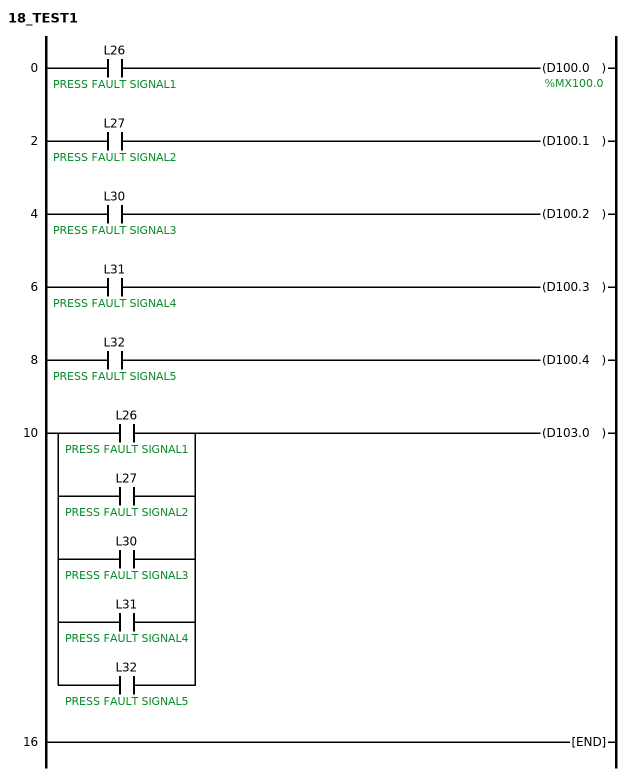
[picture p312: ladder of 18_TEST1, rungs at steps 0 to 16]
0     LD      L26  ; PRESS FAULT SIGNAL1
      OUT     D100.0  ; %MX100.0
2     LD      L27  ; PRESS FAULT SIGNAL2
      OUT     D100.1
4     LD      L30  ; PRESS FAULT SIGNAL3
      OUT     D100.2
6     LD      L31  ; PRESS FAULT SIGNAL4
      OUT     D100.3
8     LD      L32  ; PRESS FAULT SIGNAL5
      OUT     D100.4
10    LD      L26  ; PRESS FAULT SIGNAL1
      OR      L27  ; PRESS FAULT SIGNAL2
      OR      L30  ; PRESS FAULT SIGNAL3
      OR      L31  ; PRESS FAULT SIGNAL4
      OR      L32  ; PRESS FAULT SIGNAL5
      OUT     D103.0
16    END
END_PROGRAM

PROGRAM Map
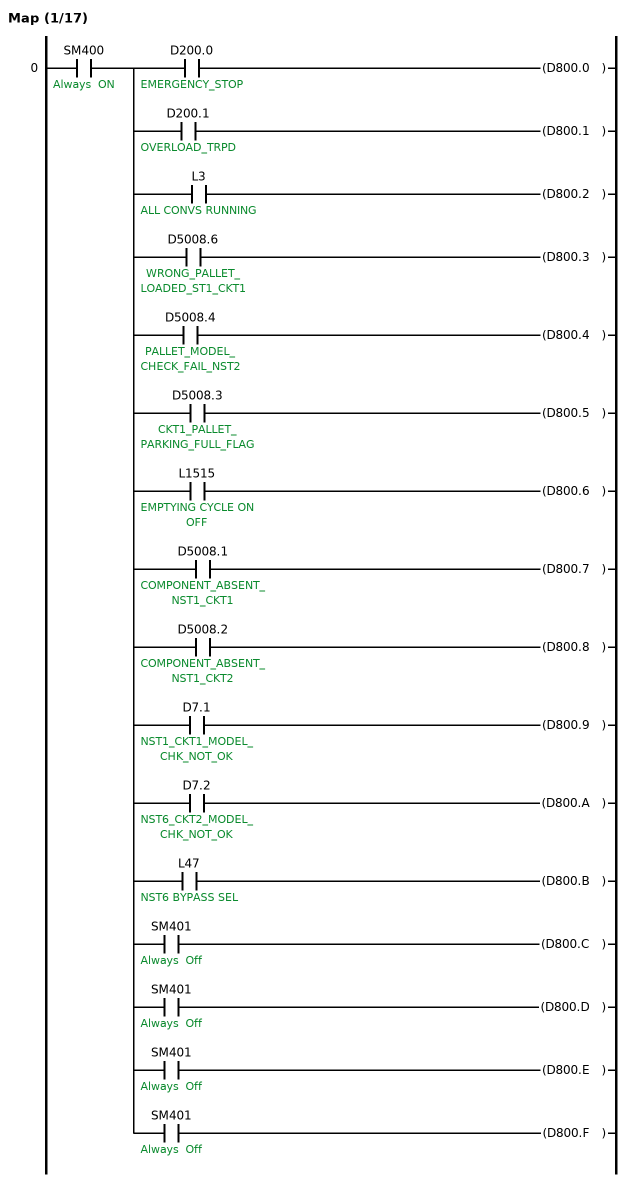
0     LD      SM400  ; Always  ON
      MPS
      AND     D200.0  ; EMERGENCY_STOP
      OUT     D800.0
      MRD
      AND     D200.1  ; OVERLOAD_TRPD
      OUT     D800.1
      MRD
      AND     L3  ; ALL CONVS RUNNING
      OUT     D800.2
      MRD
      AND     D5008.6  ; WRONG_PALLET_LOADED_ST1_CKT1
      OUT     D800.3
      MRD
      AND     D5008.4  ; PALLET_MODEL_CHECK_FAIL_NST2
      OUT     D800.4
      MRD
      AND     D5008.3  ; CKT1_PALLET_PARKING_FULL_FLAG
      OUT     D800.5
      MRD
      AND     L1515  ; EMPTYING CYCLE ON OFF
      OUT     D800.6
      MRD
      AND     D5008.1  ; COMPONENT_ABSENT_NST1_CKT1
      OUT     D800.7
      MRD
      AND     D5008.2  ; COMPONENT_ABSENT_NST1_CKT2
      OUT     D800.8
      MRD
      AND     D7.1  ; NST1_CKT1_MODEL_CHK_NOT_OK
      OUT     D800.9
      MRD
      AND     D7.2  ; NST6_CKT2_MODEL_CHK_NOT_OK
      OUT     D800.A
      MRD
      AND     L47  ; NST6 BYPASS SEL
      OUT     D800.B
      MRD
      AND     SM401  ; Always  Off
      OUT     D800.C
      MRD
      AND     SM401  ; Always  Off
      OUT     D800.D
      MRD
      AND     SM401  ; Always  Off
      OUT     D800.E
      MPP
      AND     SM401  ; Always  Off
      OUT     D800.F
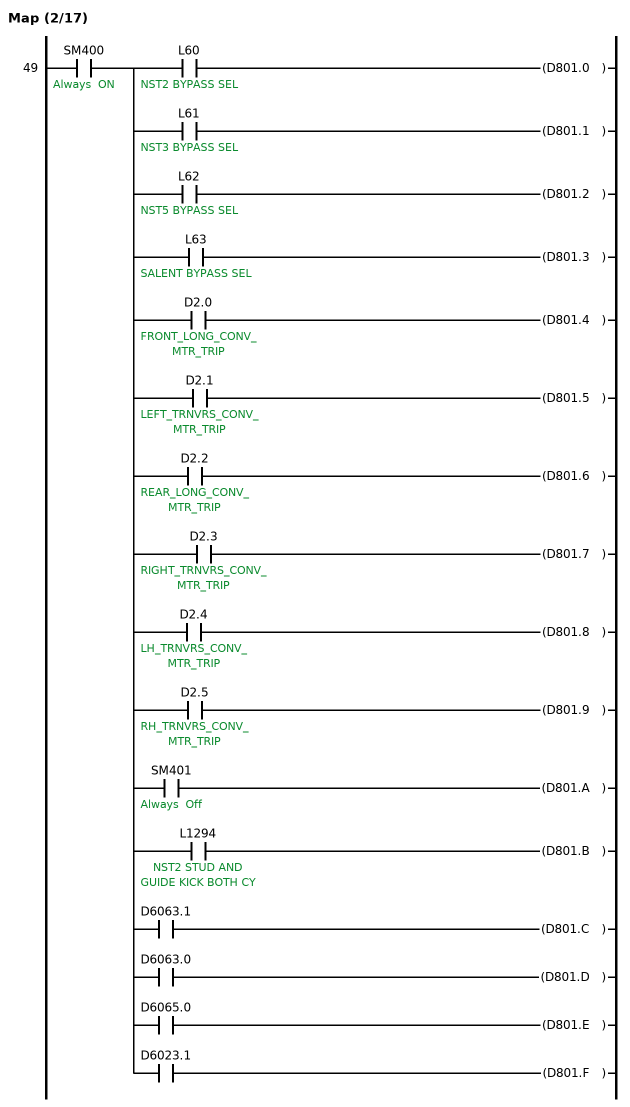
49    LD      SM400  ; Always  ON
      MPS
      AND     L60  ; NST2 BYPASS SEL
      OUT     D801.0
      MRD
      AND     L61  ; NST3 BYPASS SEL
      OUT     D801.1
      MRD
      AND     L62  ; NST5 BYPASS SEL
      OUT     D801.2
      MRD
      AND     L63  ; SALENT BYPASS SEL
      OUT     D801.3
      MRD
      AND     D2.0  ; FRONT_LONG_CONV_MTR_TRIP
      OUT     D801.4
      MRD
      AND     D2.1  ; LEFT_TRNVRS_CONV_MTR_TRIP
      OUT     D801.5
      MRD
      AND     D2.2  ; REAR_LONG_CONV_MTR_TRIP
      OUT     D801.6
      MRD
      AND     D2.3  ; RIGHT_TRNVRS_CONV_MTR_TRIP
      OUT     D801.7
      MRD
      AND     D2.4  ; LH_TRNVRS_CONV_MTR_TRIP
      OUT     D801.8
      MRD
      AND     D2.5  ; RH_TRNVRS_CONV_MTR_TRIP
      OUT     D801.9
      MRD
      AND     SM401  ; Always  Off
      OUT     D801.A
      MRD
      AND     L1294  ; NST2 STUD AND GUIDE KICK BOTH CY
      OUT     D801.B
      MRD
      AND     D6063.1
      OUT     D801.C
      MRD
      AND     D6063.0
      OUT     D801.D
      MRD
      AND     D6065.0
      OUT     D801.E
      MPP
      AND     D6023.1
      OUT     D801.F
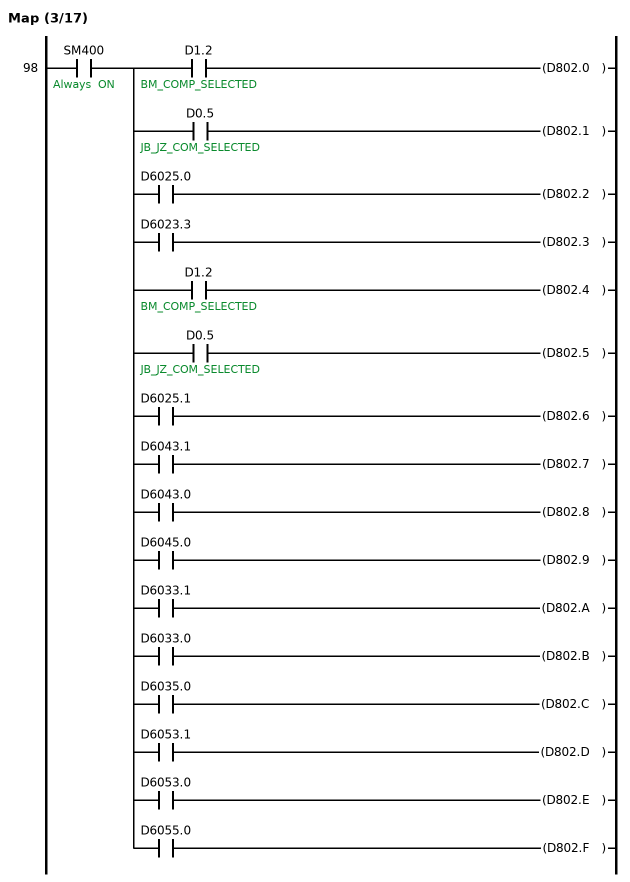
98    LD      SM400  ; Always  ON
      MPS
      AND     D1.2  ; BM_COMP_SELECTED
      OUT     D802.0
      MRD
      AND     D0.5  ; JB_JZ_COM_SELECTED
      OUT     D802.1
      MRD
      AND     D6025.0
      OUT     D802.2
      MRD
      AND     D6023.3
      OUT     D802.3
      MRD
      AND     D1.2  ; BM_COMP_SELECTED
      OUT     D802.4
      MRD
      AND     D0.5  ; JB_JZ_COM_SELECTED
      OUT     D802.5
      MRD
      AND     D6025.1
      OUT     D802.6
      MRD
      AND     D6043.1
      OUT     D802.7
      MRD
      AND     D6043.0
      OUT     D802.8
      MRD
      AND     D6045.0
      OUT     D802.9
      MRD
      AND     D6033.1
      OUT     D802.A
      MRD
      AND     D6033.0
      OUT     D802.B
      MRD
      AND     D6035.0
      OUT     D802.C
      MRD
      AND     D6053.1
      OUT     D802.D
      MRD
      AND     D6053.0
      OUT     D802.E
      MPP
      AND     D6055.0
      OUT     D802.F
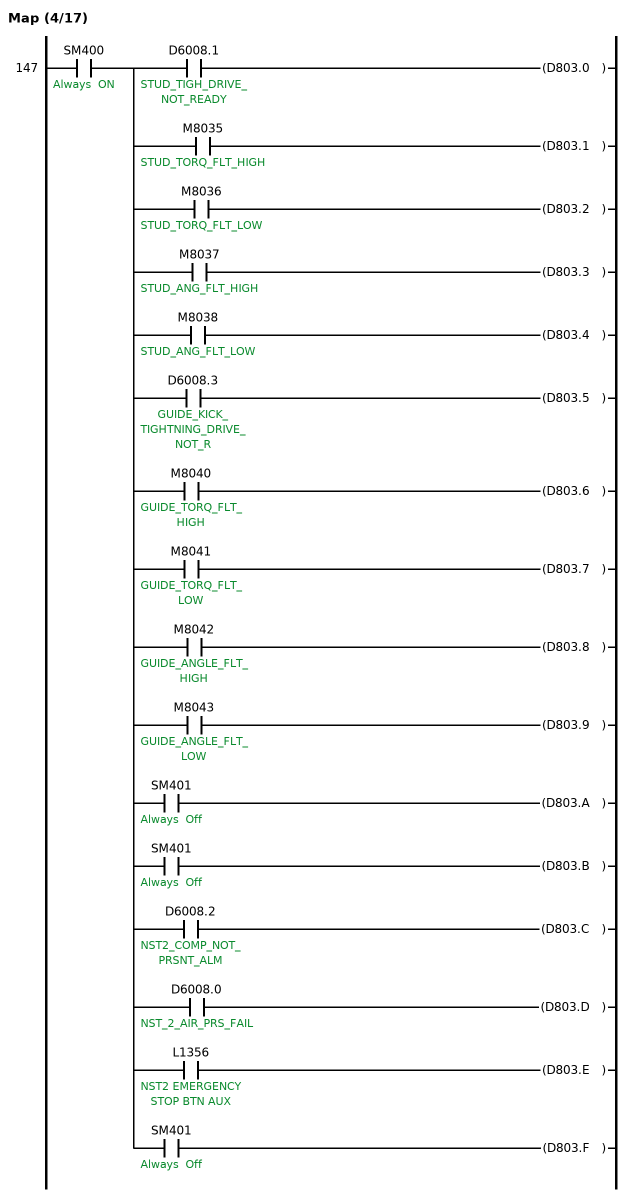
147   LD      SM400  ; Always  ON
      MPS
      AND     D6008.1  ; STUD_TIGH_DRIVE_NOT_READY
      OUT     D803.0
      MRD
      AND     M8035  ; STUD_TORQ_FLT_HIGH
      OUT     D803.1
      MRD
      AND     M8036  ; STUD_TORQ_FLT_LOW
      OUT     D803.2
      MRD
      AND     M8037  ; STUD_ANG_FLT_HIGH
      OUT     D803.3
      MRD
      AND     M8038  ; STUD_ANG_FLT_LOW
      OUT     D803.4
      MRD
      AND     D6008.3  ; GUIDE_KICK_TIGHTNING_DRIVE_NOT_R
      OUT     D803.5
      MRD
      AND     M8040  ; GUIDE_TORQ_FLT_HIGH
      OUT     D803.6
      MRD
      AND     M8041  ; GUIDE_TORQ_FLT_LOW
      OUT     D803.7
      MRD
      AND     M8042  ; GUIDE_ANGLE_FLT_HIGH
      OUT     D803.8
      MRD
      AND     M8043  ; GUIDE_ANGLE_FLT_LOW
      OUT     D803.9
      MRD
      AND     SM401  ; Always  Off
      OUT     D803.A
      MRD
      AND     SM401  ; Always  Off
      OUT     D803.B
      MRD
      AND     D6008.2  ; NST2_COMP_NOT_PRSNT_ALM
      OUT     D803.C
      MRD
      AND     D6008.0  ; NST_2_AIR_PRS_FAIL
      OUT     D803.D
      MRD
      AND     L1356  ; NST2 EMERGENCY STOP BTN AUX
      OUT     D803.E
      MPP
      AND     SM401  ; Always  Off
      OUT     D803.F
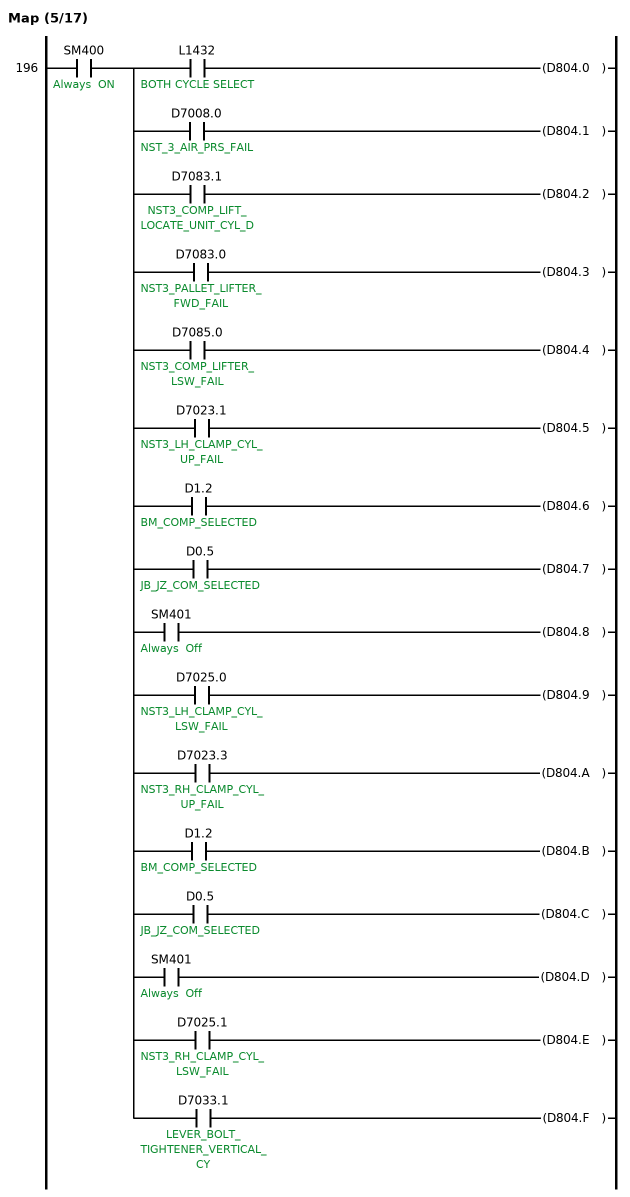
196   LD      SM400  ; Always  ON
      MPS
      AND     L1432  ; BOTH CYCLE SELECT
      OUT     D804.0
      MRD
      AND     D7008.0  ; NST_3_AIR_PRS_FAIL
      OUT     D804.1
      MRD
      AND     D7083.1  ; NST3_COMP_LIFT_LOCATE_UNIT_CYL_D
      OUT     D804.2
      MRD
      AND     D7083.0  ; NST3_PALLET_LIFTER_FWD_FAIL
      OUT     D804.3
      MRD
      AND     D7085.0  ; NST3_COMP_LIFTER_LSW_FAIL
      OUT     D804.4
      MRD
      AND     D7023.1  ; NST3_LH_CLAMP_CYL_UP_FAIL
      OUT     D804.5
      MRD
      AND     D1.2  ; BM_COMP_SELECTED
      OUT     D804.6
      MRD
      AND     D0.5  ; JB_JZ_COM_SELECTED
      OUT     D804.7
      MRD
      AND     SM401  ; Always  Off
      OUT     D804.8
      MRD
      AND     D7025.0  ; NST3_LH_CLAMP_CYL_LSW_FAIL
      OUT     D804.9
      MRD
      AND     D7023.3  ; NST3_RH_CLAMP_CYL_UP_FAIL
      OUT     D804.A
      MRD
      AND     D1.2  ; BM_COMP_SELECTED
      OUT     D804.B
      MRD
      AND     D0.5  ; JB_JZ_COM_SELECTED
      OUT     D804.C
      MRD
      AND     SM401  ; Always  Off
      OUT     D804.D
      MRD
      AND     D7025.1  ; NST3_RH_CLAMP_CYL_LSW_FAIL
      OUT     D804.E
      MPP
      AND     D7033.1  ; LEVER_BOLT_TIGHTENER_VERTICAL_CY
      OUT     D804.F
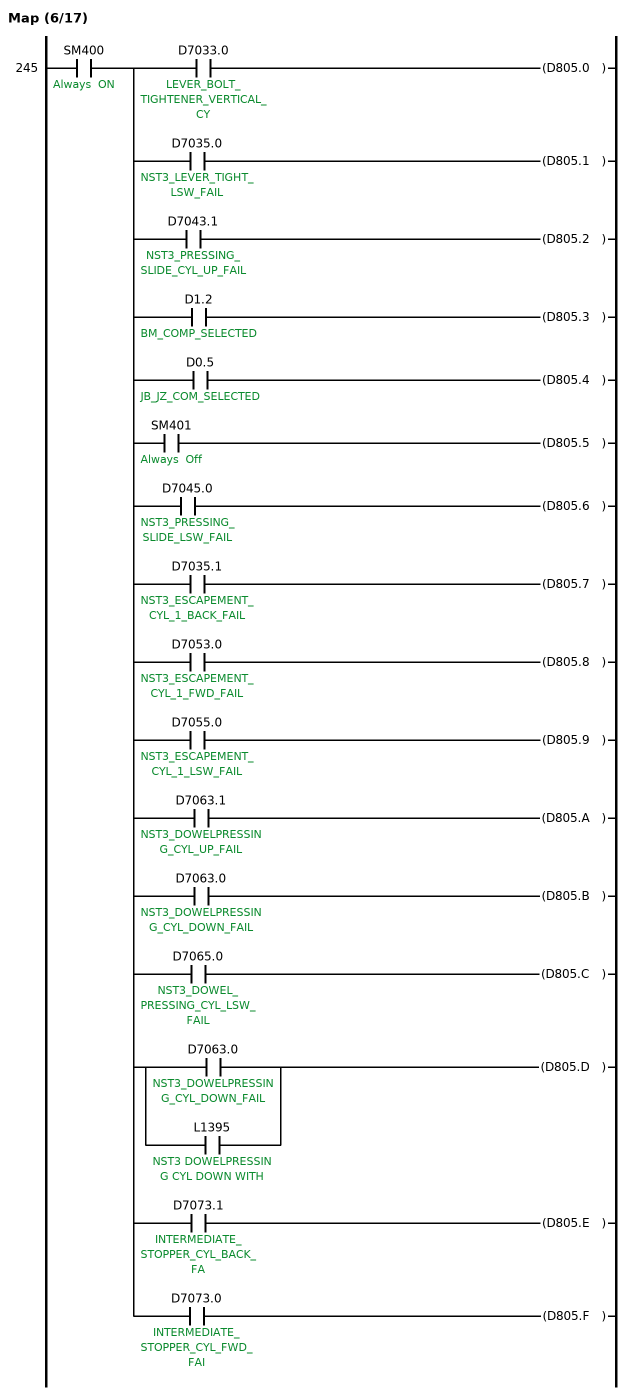
245   LD      SM400  ; Always  ON
      MPS
      AND     D7033.0  ; LEVER_BOLT_TIGHTENER_VERTICAL_CY
      OUT     D805.0
      MRD
      AND     D7035.0  ; NST3_LEVER_TIGHT_LSW_FAIL
      OUT     D805.1
      MRD
      AND     D7043.1  ; NST3_PRESSING_SLIDE_CYL_UP_FAIL
      OUT     D805.2
      MRD
      AND     D1.2  ; BM_COMP_SELECTED
      OUT     D805.3
      MRD
      AND     D0.5  ; JB_JZ_COM_SELECTED
      OUT     D805.4
      MRD
      AND     SM401  ; Always  Off
      OUT     D805.5
      MRD
      AND     D7045.0  ; NST3_PRESSING_SLIDE_LSW_FAIL
      OUT     D805.6
      MRD
      AND     D7035.1  ; NST3_ESCAPEMENT_CYL_1_BACK_FAIL
      OUT     D805.7
      MRD
      AND     D7053.0  ; NST3_ESCAPEMENT_CYL_1_FWD_FAIL
      OUT     D805.8
      MRD
      AND     D7055.0  ; NST3_ESCAPEMENT_CYL_1_LSW_FAIL
      OUT     D805.9
      MRD
      AND     D7063.1  ; NST3_DOWELPRESSING_CYL_UP_FAIL
      OUT     D805.A
      MRD
      AND     D7063.0  ; NST3_DOWELPRESSING_CYL_DOWN_FAIL
      OUT     D805.B
      MRD
      AND     D7065.0  ; NST3_DOWEL_PRESSING_CYL_LSW_FAIL
      OUT     D805.C
      MRD
      LD      D7063.0  ; NST3_DOWELPRESSING_CYL_DOWN_FAIL
      OR      L1395  ; NST3 DOWELPRESSING CYL DOWN WITH
      ANB
      OUT     D805.D
      MRD
      AND     D7073.1  ; INTERMEDIATE_STOPPER_CYL_BACK_FA
      OUT     D805.E
      MPP
      AND     D7073.0  ; INTERMEDIATE_STOPPER_CYL_FWD_FAI
      OUT     D805.F
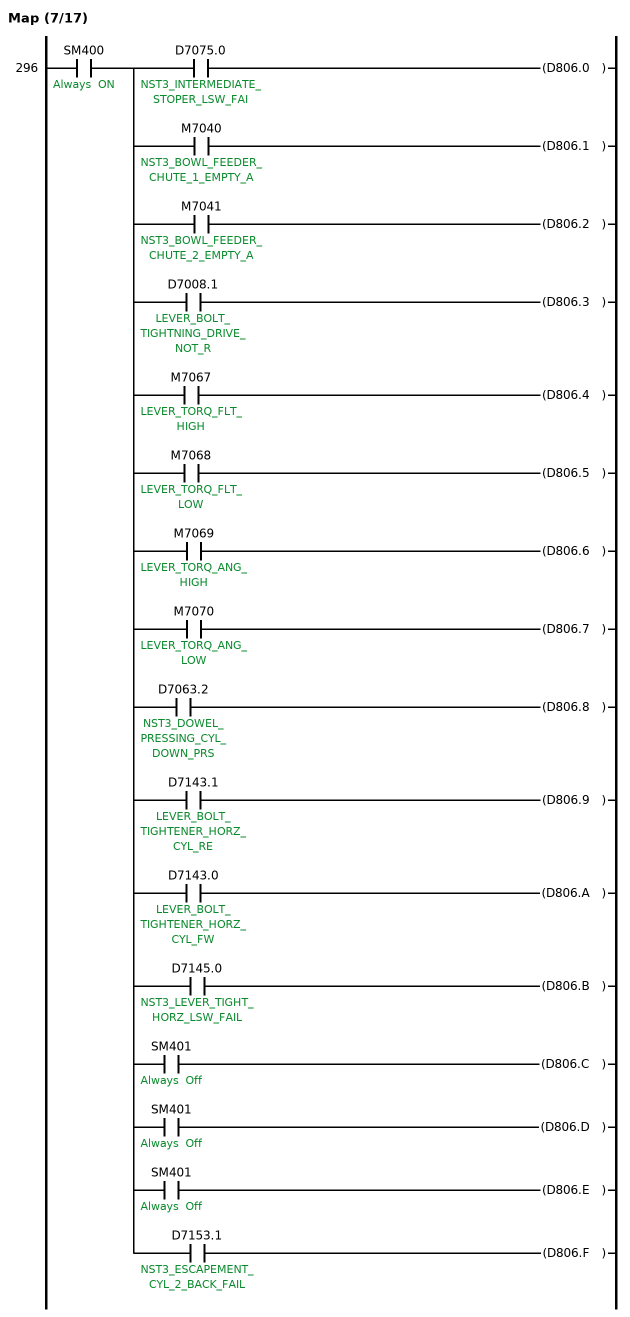
296   LD      SM400  ; Always  ON
      MPS
      AND     D7075.0  ; NST3_INTERMEDIATE_STOPER_LSW_FAI
      OUT     D806.0
      MRD
      AND     M7040  ; NST3_BOWL_FEEDER_CHUTE_1_EMPTY_A
      OUT     D806.1
      MRD
      AND     M7041  ; NST3_BOWL_FEEDER_CHUTE_2_EMPTY_A
      OUT     D806.2
      MRD
      AND     D7008.1  ; LEVER_BOLT_TIGHTNING_DRIVE_NOT_R
      OUT     D806.3
      MRD
      AND     M7067  ; LEVER_TORQ_FLT_HIGH
      OUT     D806.4
      MRD
      AND     M7068  ; LEVER_TORQ_FLT_LOW
      OUT     D806.5
      MRD
      AND     M7069  ; LEVER_TORQ_ANG_HIGH
      OUT     D806.6
      MRD
      AND     M7070  ; LEVER_TORQ_ANG_LOW
      OUT     D806.7
      MRD
      AND     D7063.2  ; NST3_DOWEL_PRESSING_CYL_DOWN_PRS
      OUT     D806.8
      MRD
      AND     D7143.1  ; LEVER_BOLT_TIGHTENER_HORZ_CYL_RE
      OUT     D806.9
      MRD
      AND     D7143.0  ; LEVER_BOLT_TIGHTENER_HORZ_CYL_FW
      OUT     D806.A
      MRD
      AND     D7145.0  ; NST3_LEVER_TIGHT_HORZ_LSW_FAIL
      OUT     D806.B
      MRD
      AND     SM401  ; Always  Off
      OUT     D806.C
      MRD
      AND     SM401  ; Always  Off
      OUT     D806.D
      MRD
      AND     SM401  ; Always  Off
      OUT     D806.E
      MPP
      AND     D7153.1  ; NST3_ESCAPEMENT_CYL_2_BACK_FAIL
      OUT     D806.F
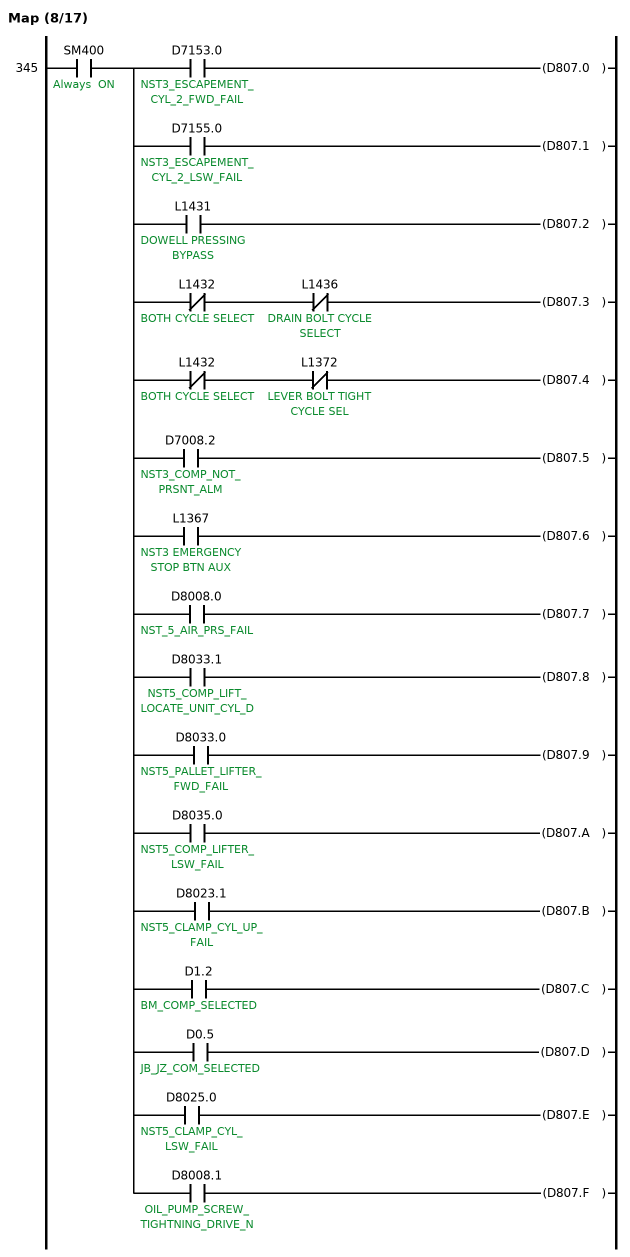
345   LD      SM400  ; Always  ON
      MPS
      AND     D7153.0  ; NST3_ESCAPEMENT_CYL_2_FWD_FAIL
      OUT     D807.0
      MRD
      AND     D7155.0  ; NST3_ESCAPEMENT_CYL_2_LSW_FAIL
      OUT     D807.1
      MRD
      AND     L1431  ; DOWELL PRESSING BYPASS
      OUT     D807.2
      MRD
      ANI     L1432  ; BOTH CYCLE SELECT
      ANI     L1436  ; DRAIN BOLT CYCLE SELECT
      OUT     D807.3
      MRD
      ANI     L1432  ; BOTH CYCLE SELECT
      ANI     L1372  ; LEVER BOLT TIGHT CYCLE SEL
      OUT     D807.4
      MRD
      AND     D7008.2  ; NST3_COMP_NOT_PRSNT_ALM
      OUT     D807.5
      MRD
      AND     L1367  ; NST3 EMERGENCY STOP BTN AUX
      OUT     D807.6
      MRD
      AND     D8008.0  ; NST_5_AIR_PRS_FAIL
      OUT     D807.7
      MRD
      AND     D8033.1  ; NST5_COMP_LIFT_LOCATE_UNIT_CYL_D
      OUT     D807.8
      MRD
      AND     D8033.0  ; NST5_PALLET_LIFTER_FWD_FAIL
      OUT     D807.9
      MRD
      AND     D8035.0  ; NST5_COMP_LIFTER_LSW_FAIL
      OUT     D807.A
      MRD
      AND     D8023.1  ; NST5_CLAMP_CYL_UP_FAIL
      OUT     D807.B
      MRD
      AND     D1.2  ; BM_COMP_SELECTED
      OUT     D807.C
      MRD
      AND     D0.5  ; JB_JZ_COM_SELECTED
      OUT     D807.D
      MRD
      AND     D8025.0  ; NST5_CLAMP_CYL_LSW_FAIL
      OUT     D807.E
      MPP
      AND     D8008.1  ; OIL_PUMP_SCREW_TIGHTNING_DRIVE_N
      OUT     D807.F
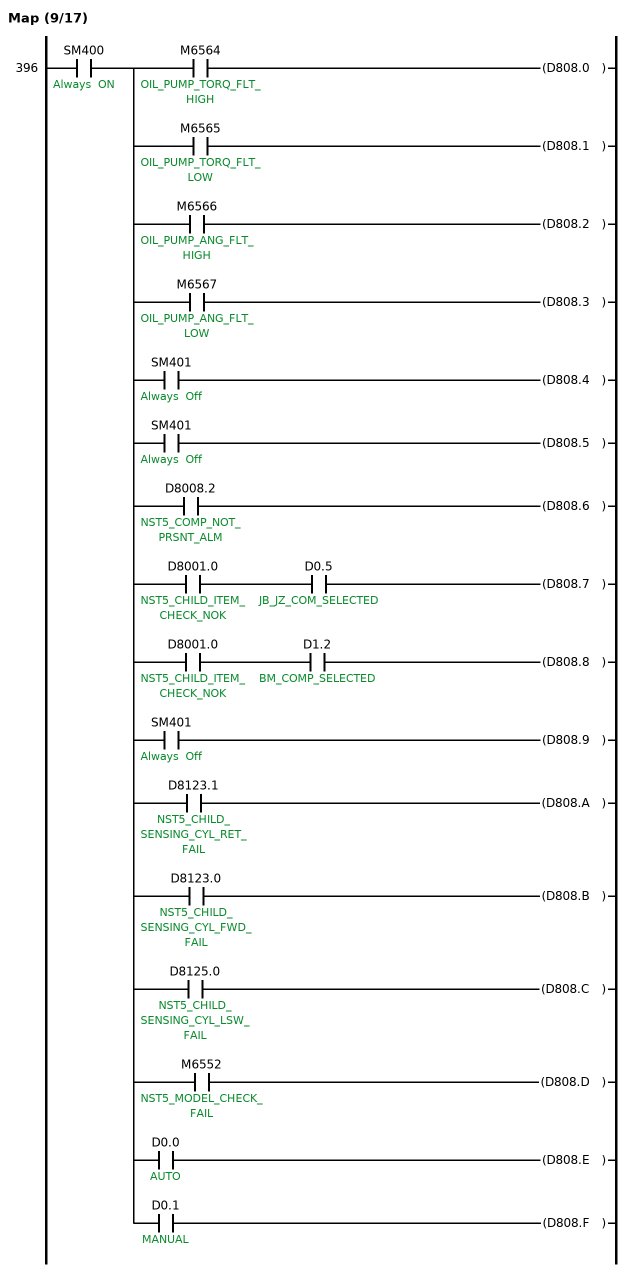
396   LD      SM400  ; Always  ON
      MPS
      AND     M6564  ; OIL_PUMP_TORQ_FLT_HIGH
      OUT     D808.0
      MRD
      AND     M6565  ; OIL_PUMP_TORQ_FLT_LOW
      OUT     D808.1
      MRD
      AND     M6566  ; OIL_PUMP_ANG_FLT_HIGH
      OUT     D808.2
      MRD
      AND     M6567  ; OIL_PUMP_ANG_FLT_LOW
      OUT     D808.3
      MRD
      AND     SM401  ; Always  Off
      OUT     D808.4
      MRD
      AND     SM401  ; Always  Off
      OUT     D808.5
      MRD
      AND     D8008.2  ; NST5_COMP_NOT_PRSNT_ALM
      OUT     D808.6
      MRD
      AND     D8001.0  ; NST5_CHILD_ITEM_CHECK_NOK
      AND     D0.5  ; JB_JZ_COM_SELECTED
      OUT     D808.7
      MRD
      AND     D8001.0  ; NST5_CHILD_ITEM_CHECK_NOK
      AND     D1.2  ; BM_COMP_SELECTED
      OUT     D808.8
      MRD
      AND     SM401  ; Always  Off
      OUT     D808.9
      MRD
      AND     D8123.1  ; NST5_CHILD_SENSING_CYL_RET_FAIL
      OUT     D808.A
      MRD
      AND     D8123.0  ; NST5_CHILD_SENSING_CYL_FWD_FAIL
      OUT     D808.B
      MRD
      AND     D8125.0  ; NST5_CHILD_SENSING_CYL_LSW_FAIL
      OUT     D808.C
      MRD
      AND     M6552  ; NST5_MODEL_CHECK_FAIL
      OUT     D808.D
      MRD
      AND     D0.0  ; AUTO
      OUT     D808.E
      MPP
      AND     D0.1  ; MANUAL
      OUT     D808.F
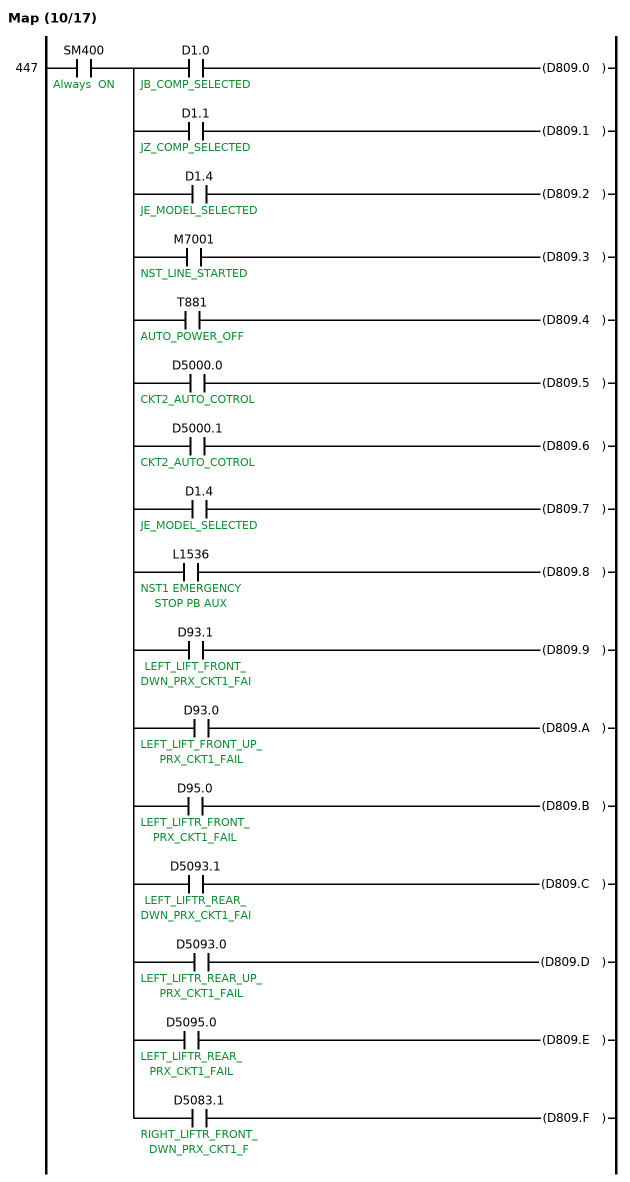
447   LD      SM400  ; Always  ON
      MPS
      AND     D1.0  ; JB_COMP_SELECTED
      OUT     D809.0
      MRD
      AND     D1.1  ; JZ_COMP_SELECTED
      OUT     D809.1
      MRD
      AND     D1.4  ; JE_MODEL_SELECTED
      OUT     D809.2
      MRD
      AND     M7001  ; NST_LINE_STARTED
      OUT     D809.3
      MRD
      AND     T881  ; AUTO_POWER_OFF
      OUT     D809.4
      MRD
      AND     D5000.0  ; CKT2_AUTO_COTROL
      OUT     D809.5
      MRD
      AND     D5000.1  ; CKT2_AUTO_COTROL
      OUT     D809.6
      MRD
      AND     D1.4  ; JE_MODEL_SELECTED
      OUT     D809.7
      MRD
      AND     L1536  ; NST1 EMERGENCY STOP PB AUX
      OUT     D809.8
      MRD
      AND     D93.1  ; LEFT_LIFT_FRONT_DWN_PRX_CKT1_FAI
      OUT     D809.9
      MRD
      AND     D93.0  ; LEFT_LIFT_FRONT_UP_PRX_CKT1_FAIL
      OUT     D809.A
      MRD
      AND     D95.0  ; LEFT_LIFTR_FRONT_PRX_CKT1_FAIL
      OUT     D809.B
      MRD
      AND     D5093.1  ; LEFT_LIFTR_REAR_DWN_PRX_CKT1_FAI
      OUT     D809.C
      MRD
      AND     D5093.0  ; LEFT_LIFTR_REAR_UP_PRX_CKT1_FAIL
      OUT     D809.D
      MRD
      AND     D5095.0  ; LEFT_LIFTR_REAR_PRX_CKT1_FAIL
      OUT     D809.E
      MPP
      AND     D5083.1  ; RIGHT_LIFTR_FRONT_DWN_PRX_CKT1_F
      OUT     D809.F
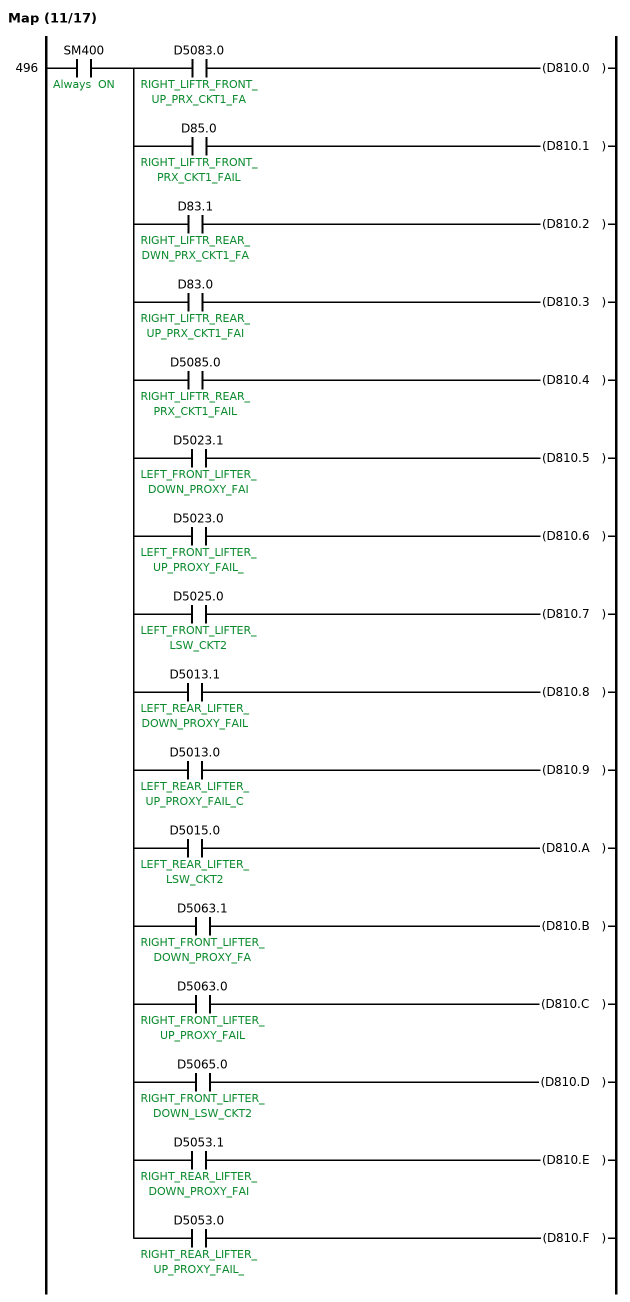
496   LD      SM400  ; Always  ON
      MPS
      AND     D5083.0  ; RIGHT_LIFTR_FRONT_UP_PRX_CKT1_FA
      OUT     D810.0
      MRD
      AND     D85.0  ; RIGHT_LIFTR_FRONT_PRX_CKT1_FAIL
      OUT     D810.1
      MRD
      AND     D83.1  ; RIGHT_LIFTR_REAR_DWN_PRX_CKT1_FA
      OUT     D810.2
      MRD
      AND     D83.0  ; RIGHT_LIFTR_REAR_UP_PRX_CKT1_FAI
      OUT     D810.3
      MRD
      AND     D5085.0  ; RIGHT_LIFTR_REAR_PRX_CKT1_FAIL
      OUT     D810.4
      MRD
      AND     D5023.1  ; LEFT_FRONT_LIFTER_DOWN_PROXY_FAI
      OUT     D810.5
      MRD
      AND     D5023.0  ; LEFT_FRONT_LIFTER_UP_PROXY_FAIL_
      OUT     D810.6
      MRD
      AND     D5025.0  ; LEFT_FRONT_LIFTER_LSW_CKT2
      OUT     D810.7
      MRD
      AND     D5013.1  ; LEFT_REAR_LIFTER_DOWN_PROXY_FAIL
      OUT     D810.8
      MRD
      AND     D5013.0  ; LEFT_REAR_LIFTER_UP_PROXY_FAIL_C
      OUT     D810.9
      MRD
      AND     D5015.0  ; LEFT_REAR_LIFTER_LSW_CKT2
      OUT     D810.A
      MRD
      AND     D5063.1  ; RIGHT_FRONT_LIFTER_DOWN_PROXY_FA
      OUT     D810.B
      MRD
      AND     D5063.0  ; RIGHT_FRONT_LIFTER_UP_PROXY_FAIL
      OUT     D810.C
      MRD
      AND     D5065.0  ; RIGHT_FRONT_LIFTER_DOWN_LSW_CKT2
      OUT     D810.D
      MRD
      AND     D5053.1  ; RIGHT_REAR_LIFTER_DOWN_PROXY_FAI
      OUT     D810.E
      MPP
      AND     D5053.0  ; RIGHT_REAR_LIFTER_UP_PROXY_FAIL_
      OUT     D810.F
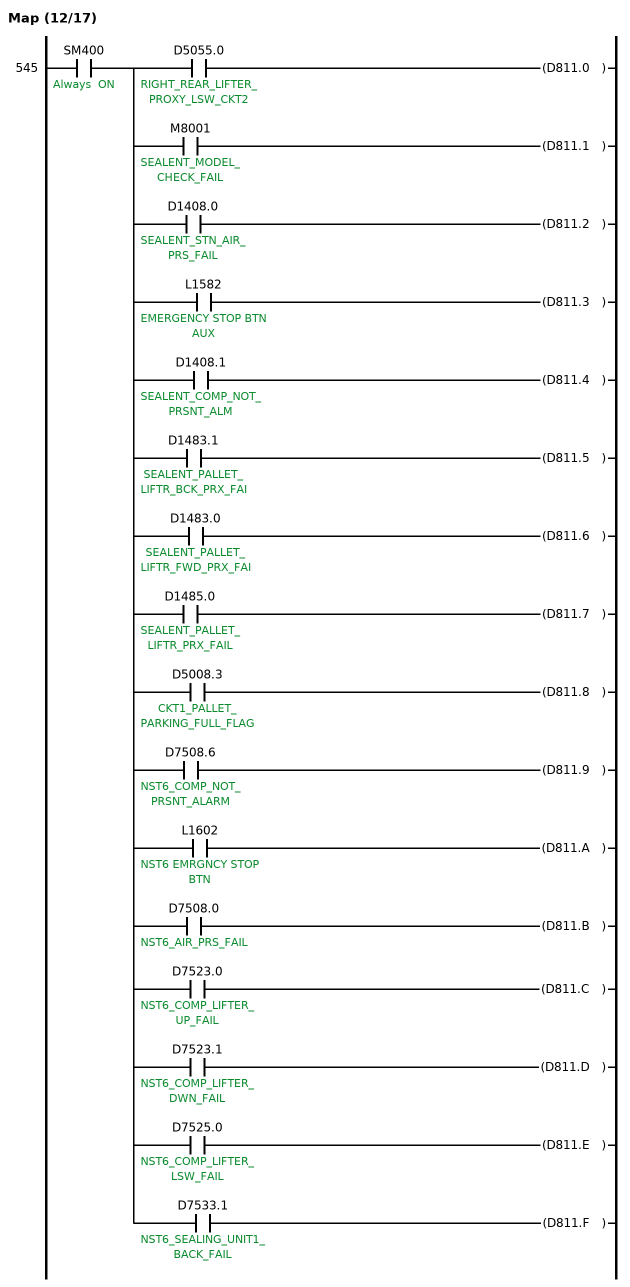
545   LD      SM400  ; Always  ON
      MPS
      AND     D5055.0  ; RIGHT_REAR_LIFTER_PROXY_LSW_CKT2
      OUT     D811.0
      MRD
      AND     M8001  ; SEALENT_MODEL_CHECK_FAIL
      OUT     D811.1
      MRD
      AND     D1408.0  ; SEALENT_STN_AIR_PRS_FAIL
      OUT     D811.2
      MRD
      AND     L1582  ; EMERGENCY STOP BTN AUX
      OUT     D811.3
      MRD
      AND     D1408.1  ; SEALENT_COMP_NOT_PRSNT_ALM
      OUT     D811.4
      MRD
      AND     D1483.1  ; SEALENT_PALLET_LIFTR_BCK_PRX_FAI
      OUT     D811.5
      MRD
      AND     D1483.0  ; SEALENT_PALLET_LIFTR_FWD_PRX_FAI
      OUT     D811.6
      MRD
      AND     D1485.0  ; SEALENT_PALLET_LIFTR_PRX_FAIL
      OUT     D811.7
      MRD
      AND     D5008.3  ; CKT1_PALLET_PARKING_FULL_FLAG
      OUT     D811.8
      MRD
      AND     D7508.6  ; NST6_COMP_NOT_PRSNT_ALARM
      OUT     D811.9
      MRD
      AND     L1602  ; NST6 EMRGNCY STOP BTN
      OUT     D811.A
      MRD
      AND     D7508.0  ; NST6_AIR_PRS_FAIL
      OUT     D811.B
      MRD
      AND     D7523.0  ; NST6_COMP_LIFTER_UP_FAIL
      OUT     D811.C
      MRD
      AND     D7523.1  ; NST6_COMP_LIFTER_DWN_FAIL
      OUT     D811.D
      MRD
      AND     D7525.0  ; NST6_COMP_LIFTER_LSW_FAIL
      OUT     D811.E
      MPP
      AND     D7533.1  ; NST6_SEALING_UNIT1_BACK_FAIL
      OUT     D811.F
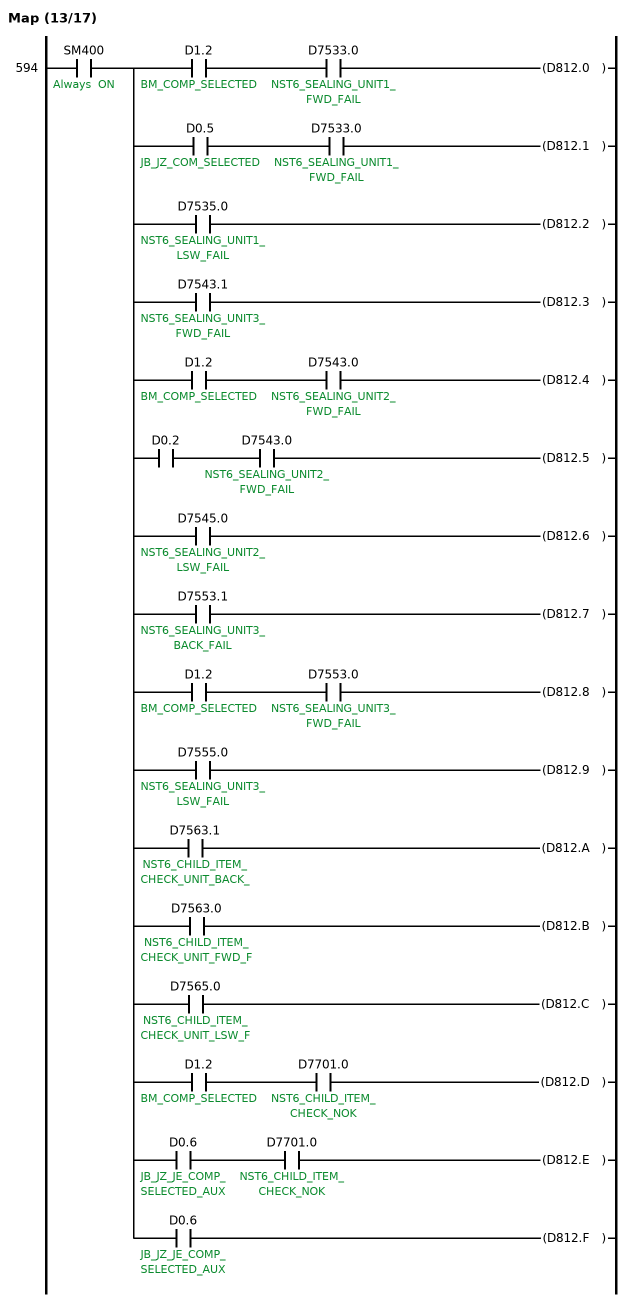
594   LD      SM400  ; Always  ON
      MPS
      AND     D1.2  ; BM_COMP_SELECTED
      AND     D7533.0  ; NST6_SEALING_UNIT1_FWD_FAIL
      OUT     D812.0
      MRD
      AND     D0.5  ; JB_JZ_COM_SELECTED
      AND     D7533.0  ; NST6_SEALING_UNIT1_FWD_FAIL
      OUT     D812.1
      MRD
      AND     D7535.0  ; NST6_SEALING_UNIT1_LSW_FAIL
      OUT     D812.2
      MRD
      AND     D7543.1  ; NST6_SEALING_UNIT3_FWD_FAIL
      OUT     D812.3
      MRD
      AND     D1.2  ; BM_COMP_SELECTED
      AND     D7543.0  ; NST6_SEALING_UNIT2_FWD_FAIL
      OUT     D812.4
      MRD
      AND     D0.2
      AND     D7543.0  ; NST6_SEALING_UNIT2_FWD_FAIL
      OUT     D812.5
      MRD
      AND     D7545.0  ; NST6_SEALING_UNIT2_LSW_FAIL
      OUT     D812.6
      MRD
      AND     D7553.1  ; NST6_SEALING_UNIT3_BACK_FAIL
      OUT     D812.7
      MRD
      AND     D1.2  ; BM_COMP_SELECTED
      AND     D7553.0  ; NST6_SEALING_UNIT3_FWD_FAIL
      OUT     D812.8
      MRD
      AND     D7555.0  ; NST6_SEALING_UNIT3_LSW_FAIL
      OUT     D812.9
      MRD
      AND     D7563.1  ; NST6_CHILD_ITEM_CHECK_UNIT_BACK_
      OUT     D812.A
      MRD
      AND     D7563.0  ; NST6_CHILD_ITEM_CHECK_UNIT_FWD_F
      OUT     D812.B
      MRD
      AND     D7565.0  ; NST6_CHILD_ITEM_CHECK_UNIT_LSW_F
      OUT     D812.C
      MRD
      AND     D1.2  ; BM_COMP_SELECTED
      AND     D7701.0  ; NST6_CHILD_ITEM_CHECK_NOK
      OUT     D812.D
      MRD
      AND     D0.6  ; JB_JZ_JE_COMP_SELECTED_AUX
      AND     D7701.0  ; NST6_CHILD_ITEM_CHECK_NOK
      OUT     D812.E
      MPP
      AND     D0.6  ; JB_JZ_JE_COMP_SELECTED_AUX
      OUT     D812.F
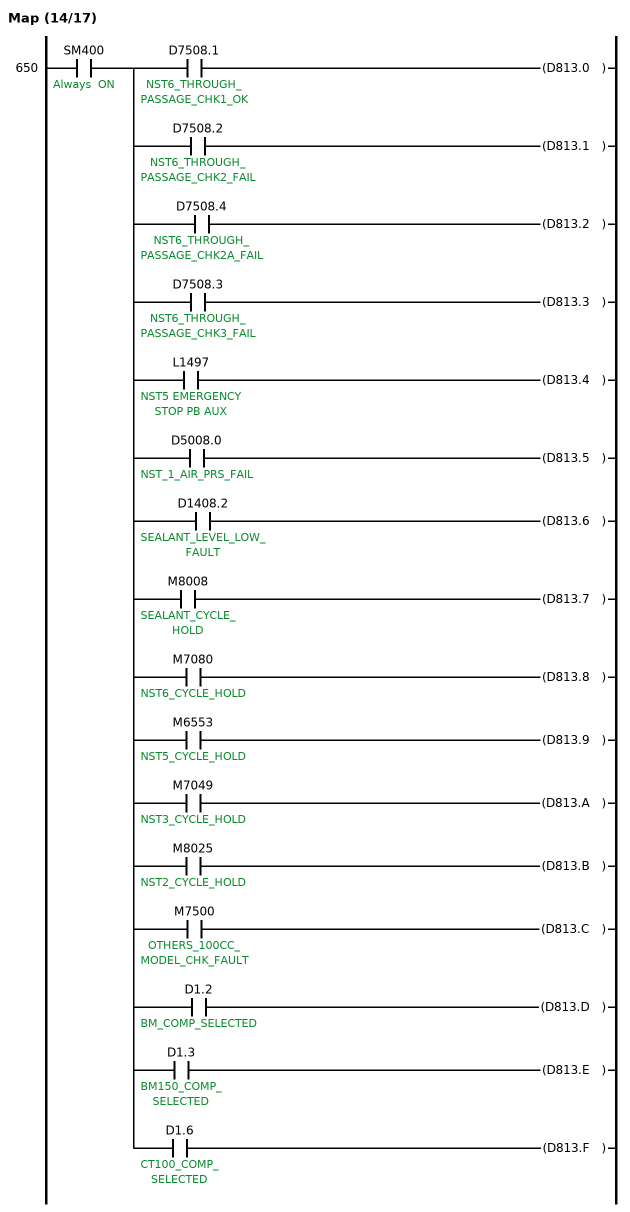
650   LD      SM400  ; Always  ON
      MPS
      AND     D7508.1  ; NST6_THROUGH_PASSAGE_CHK1_OK
      OUT     D813.0
      MRD
      AND     D7508.2  ; NST6_THROUGH_PASSAGE_CHK2_FAIL
      OUT     D813.1
      MRD
      AND     D7508.4  ; NST6_THROUGH_PASSAGE_CHK2A_FAIL
      OUT     D813.2
      MRD
      AND     D7508.3  ; NST6_THROUGH_PASSAGE_CHK3_FAIL
      OUT     D813.3
      MRD
      AND     L1497  ; NST5 EMERGENCY STOP PB AUX
      OUT     D813.4
      MRD
      AND     D5008.0  ; NST_1_AIR_PRS_FAIL
      OUT     D813.5
      MRD
      AND     D1408.2  ; SEALANT_LEVEL_LOW_FAULT
      OUT     D813.6
      MRD
      AND     M8008  ; SEALANT_CYCLE_HOLD
      OUT     D813.7
      MRD
      AND     M7080  ; NST6_CYCLE_HOLD
      OUT     D813.8
      MRD
      AND     M6553  ; NST5_CYCLE_HOLD
      OUT     D813.9
      MRD
      AND     M7049  ; NST3_CYCLE_HOLD
      OUT     D813.A
      MRD
      AND     M8025  ; NST2_CYCLE_HOLD
      OUT     D813.B
      MRD
      AND     M7500  ; OTHERS_100CC_MODEL_CHK_FAULT
      OUT     D813.C
      MRD
      AND     D1.2  ; BM_COMP_SELECTED
      OUT     D813.D
      MRD
      AND     D1.3  ; BM150_COMP_SELECTED
      OUT     D813.E
      MPP
      AND     D1.6  ; CT100_COMP_SELECTED
      OUT     D813.F
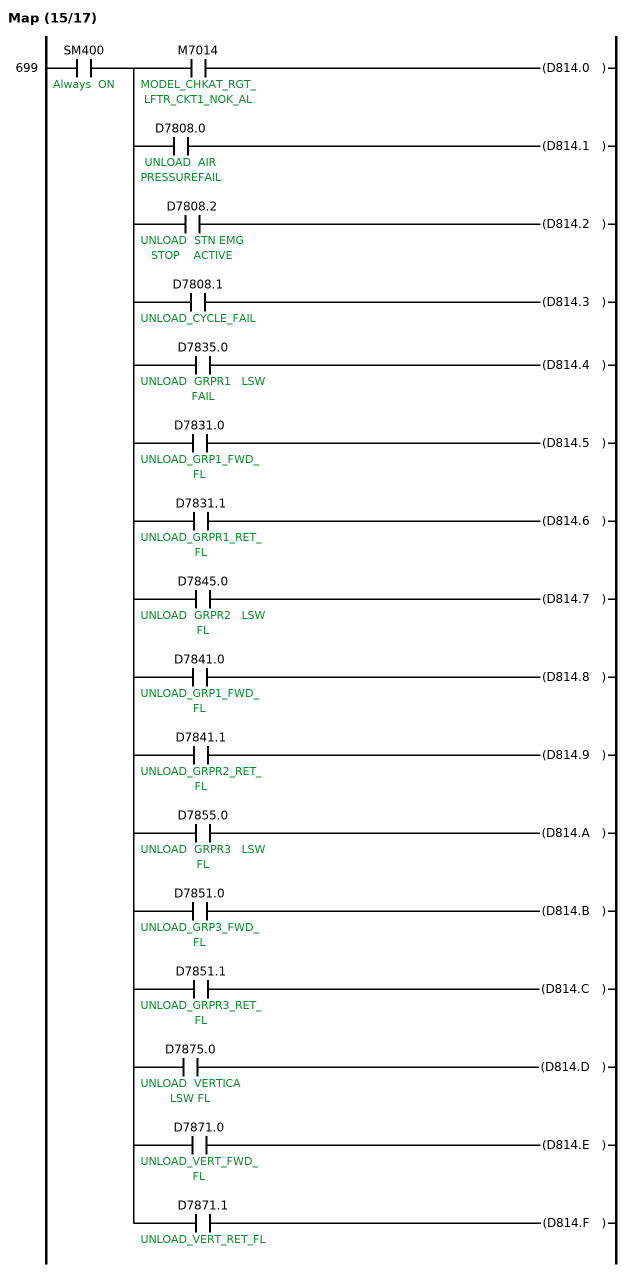
699   LD      SM400  ; Always  ON
      MPS
      AND     M7014  ; MODEL_CHKAT_RGT_LFTR_CKT1_NOK_AL
      OUT     D814.0
      MRD
      AND     D7808.0  ; UNLOAD  AIR     PRESSUREFAIL
      OUT     D814.1
      MRD
      AND     D7808.2  ; UNLOAD  STN EMG STOP    ACTIVE
      OUT     D814.2
      MRD
      AND     D7808.1  ; UNLOAD_CYCLE_FAIL
      OUT     D814.3
      MRD
      AND     D7835.0  ; UNLOAD  GRPR1   LSW FAIL
      OUT     D814.4
      MRD
      AND     D7831.0  ; UNLOAD_GRP1_FWD_FL
      OUT     D814.5
      MRD
      AND     D7831.1  ; UNLOAD_GRPR1_RET_FL
      OUT     D814.6
      MRD
      AND     D7845.0  ; UNLOAD  GRPR2   LSW FL
      OUT     D814.7
      MRD
      AND     D7841.0  ; UNLOAD_GRP1_FWD_FL
      OUT     D814.8
      MRD
      AND     D7841.1  ; UNLOAD_GRPR2_RET_FL
      OUT     D814.9
      MRD
      AND     D7855.0  ; UNLOAD  GRPR3   LSW FL
      OUT     D814.A
      MRD
      AND     D7851.0  ; UNLOAD_GRP3_FWD_FL
      OUT     D814.B
      MRD
      AND     D7851.1  ; UNLOAD_GRPR3_RET_FL
      OUT     D814.C
      MRD
      AND     D7875.0  ; UNLOAD  VERTICA LSW FL
      OUT     D814.D
      MRD
      AND     D7871.0  ; UNLOAD_VERT_FWD_FL
      OUT     D814.E
      MPP
      AND     D7871.1  ; UNLOAD_VERT_RET_FL
      OUT     D814.F
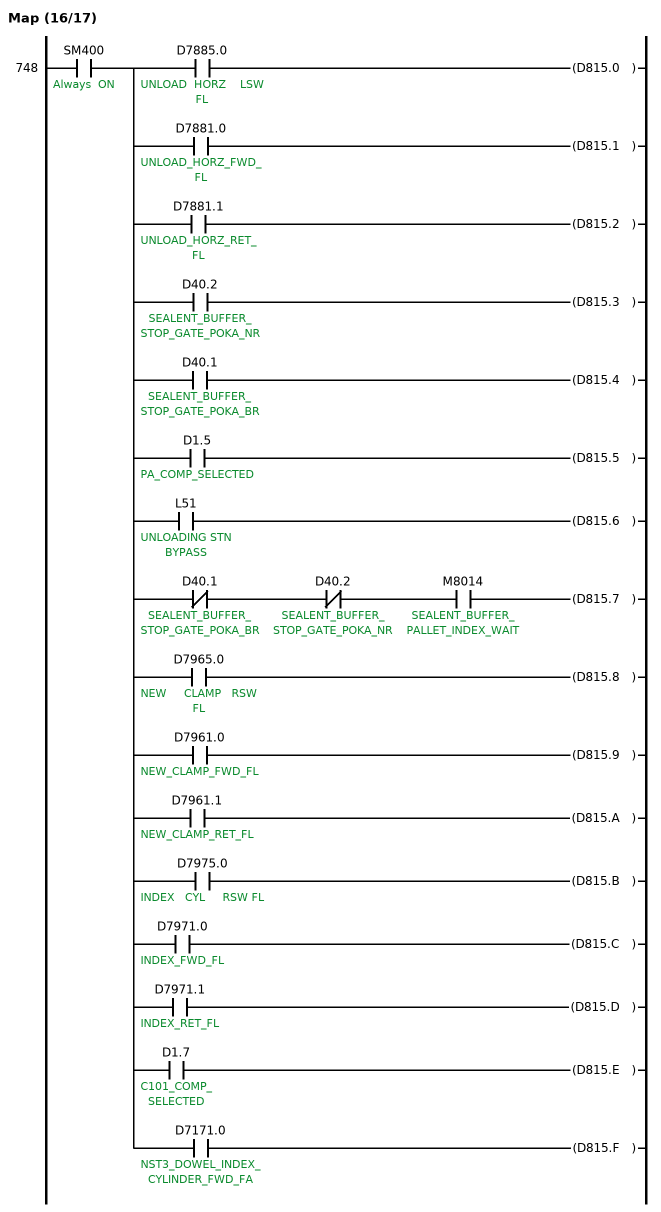
748   LD      SM400  ; Always  ON
      MPS
      AND     D7885.0  ; UNLOAD  HORZ    LSW FL
      OUT     D815.0
      MRD
      AND     D7881.0  ; UNLOAD_HORZ_FWD_FL
      OUT     D815.1
      MRD
      AND     D7881.1  ; UNLOAD_HORZ_RET_FL
      OUT     D815.2
      MRD
      AND     D40.2  ; SEALENT_BUFFER_STOP_GATE_POKA_NR
      OUT     D815.3
      MRD
      AND     D40.1  ; SEALENT_BUFFER_STOP_GATE_POKA_BR
      OUT     D815.4
      MRD
      AND     D1.5  ; PA_COMP_SELECTED
      OUT     D815.5
      MRD
      AND     L51  ; UNLOADING STN BYPASS
      OUT     D815.6
      MRD
      ANI     D40.1  ; SEALENT_BUFFER_STOP_GATE_POKA_BR
      ANI     D40.2  ; SEALENT_BUFFER_STOP_GATE_POKA_NR
      AND     M8014  ; SEALENT_BUFFER_PALLET_INDEX_WAIT
      OUT     D815.7
      MRD
      AND     D7965.0  ; NEW     CLAMP   RSW FL
      OUT     D815.8
      MRD
      AND     D7961.0  ; NEW_CLAMP_FWD_FL
      OUT     D815.9
      MRD
      AND     D7961.1  ; NEW_CLAMP_RET_FL
      OUT     D815.A
      MRD
      AND     D7975.0  ; INDEX   CYL     RSW FL
      OUT     D815.B
      MRD
      AND     D7971.0  ; INDEX_FWD_FL
      OUT     D815.C
      MRD
      AND     D7971.1  ; INDEX_RET_FL
      OUT     D815.D
      MRD
      AND     D1.7  ; C101_COMP_SELECTED
      OUT     D815.E
      MPP
      AND     D7171.0  ; NST3_DOWEL_INDEX_CYLINDER_FWD_FA
      OUT     D815.F
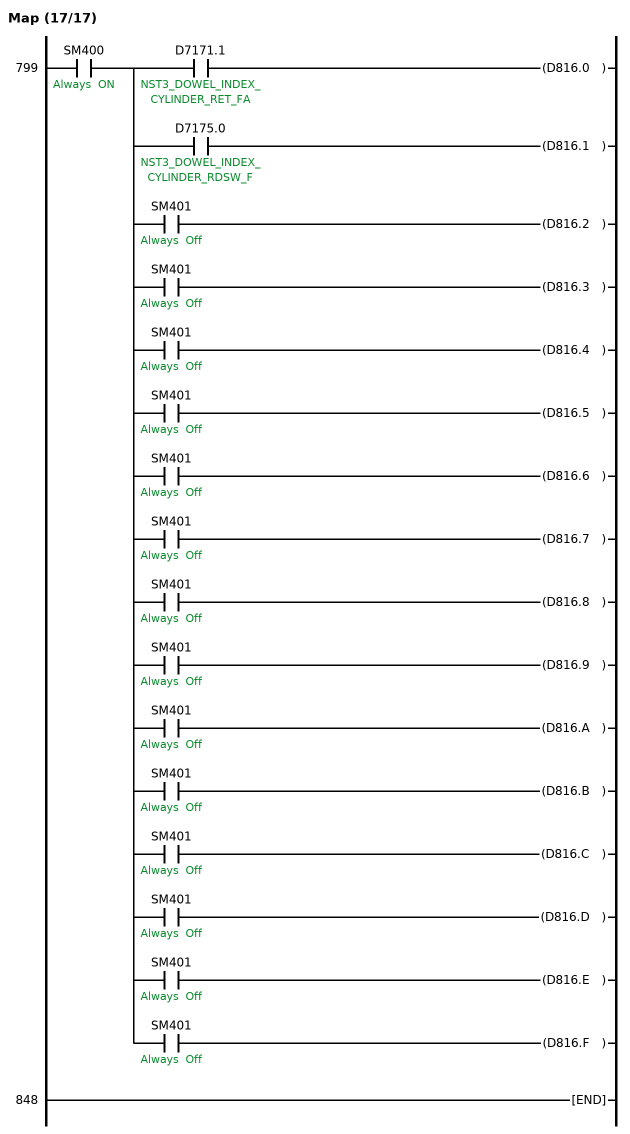
799   LD      SM400  ; Always  ON
      MPS
      AND     D7171.1  ; NST3_DOWEL_INDEX_CYLINDER_RET_FA
      OUT     D816.0
      MRD
      AND     D7175.0  ; NST3_DOWEL_INDEX_CYLINDER_RDSW_F
      OUT     D816.1
      MRD
      AND     SM401  ; Always  Off
      OUT     D816.2
      MRD
      AND     SM401  ; Always  Off
      OUT     D816.3
      MRD
      AND     SM401  ; Always  Off
      OUT     D816.4
      MRD
      AND     SM401  ; Always  Off
      OUT     D816.5
      MRD
      AND     SM401  ; Always  Off
      OUT     D816.6
      MRD
      AND     SM401  ; Always  Off
      OUT     D816.7
      MRD
      AND     SM401  ; Always  Off
      OUT     D816.8
      MRD
      AND     SM401  ; Always  Off
      OUT     D816.9
      MRD
      AND     SM401  ; Always  Off
      OUT     D816.A
      MRD
      AND     SM401  ; Always  Off
      OUT     D816.B
      MRD
      AND     SM401  ; Always  Off
      OUT     D816.C
      MRD
      AND     SM401  ; Always  Off
      OUT     D816.D
      MRD
      AND     SM401  ; Always  Off
      OUT     D816.E
      MPP
      AND     SM401  ; Always  Off
      OUT     D816.F
848   END
END_PROGRAM

// device comments not shown above
L22  ; N1 883 CYC CMPLT SIGNAL
L25  ; N1 882 CYC CMPLT SIGNAL
L37  ; UNLOAD MACHINE GATE CKT1 PALLET
L77  ; COMP PRESENT AT UNLOADING STN CK
L1357  ; NST2 DRAIN BOLT SENSOR AT BUFFER
L1398  ; NST3 ESCAPEMENT CYL 2 FWD RS
L1399  ; NST3 LH CLAMP CYL DOWN RS CT100
L1493  ; NST5 MODEL IDENTIFICATION SENSOR
L1672  ; COMP PRESENT AT OUTLET OF CONV
L1673  ; UNLOADING CONV INDEX SENS
L1674  ; UNLOADING CONV HEALTHY SGNL
L1675  ; UNLOADING CONV HEALTHY SGNL1
F1307  ; NST2 BUFFER PALLET GATE DOWN SOL
F1315  ; STUD TIGHTENING DRIVE CONFIG 3
F1316  ; STUD TIGHTENING DRIVE CONFIG 4
F1322  ; GUIDE KICK TIGHTENING DRIVE REVE
F1357  ; LEVER BOLT TIGHTENING DRIVE CONF
F1402  ; OIL  PUMP  SCREW  TIGHTENING  DR
F1437  ; NST5  ROBO  POUSE  LAMP
F1494  ; UNLOADING GANTRY CYCLE RDY LAMP
F1495  ; UNLOADING GANTRY CYCLE RUNNING L
F1496  ; UNLOADING GANTRY STN FAULT LAMP
F1587  ; PRESSURE RELEIF VALVE
F1593  ; UNLAOD STN HEALTHY1 TO CONVEROR
M6559  ; ROBO_CYCLE_COUNT_RESET
M7060  ; NST_LINE_STARTED
M7804  ; NST_LINE_STARTEDM7001
M7805  ; SKIP
M7807  ; UNLOAD_CYCLE_HOLD
T416  ; SEALENT_COMP_NOT_PRSNT_EMPTYING_
D151.6  ; LAMP_TEST
D500.0  ; CKT2_AUTO_COTROL
D1404.5  ; SEALENT_LSW_FAIL
D7506.6  ; NST6_BLANK_COMM
D7809.2  ; UNLOAD_BLANK_COMM
D7809.8  ; UNLOAD_BLANK_COMM
